Staubli VAL3: Output.pgx

program Output(num io, bool cde)
begin
  //*******************************************************************************
  //*   ______
  //*  / _____) /|
  //* | |      / /
  //* | | /\  / /
  //* | | \ \/ /  _      Copyright (c) KEOLABS, 2016
  //* | |  \__/  | |        http://www.keolabs.com
  //* | |________| |
  //*  \__________/
  //*
  //********************************************************************************
  //*@file          : Output
  //*@author        : Yves Ragot
  //*@version       : $Id: Output.pgx 1202 2016-10-07 12:12:19Z yves $
  //*@brief         : set Output value
  //*
  //*******************************************************************************/

  switch (io)

    case 1
        call Valve(cde)
    break

    case 2
        doValve2 = cde
    break

    case 3
        doPump = cde
    break

    default
        GeneralStatus = 101
        LastErrorCode = 0
    break

  endSwitch

end
